Yaskawa INFORM job: R1_W27-A2(70,-90)ZJEBANY.JBI

/JOB
//NAME R1_W27-A2(70,-90)ZJEBANY
///FOLDERNAME KRIS-SCIANA
//POS
///NPOS 112,112,0,3,0,0
///TOOL 0
///POSTYPE PULSE
///PULSE
C00000=15585,66998,-23352,-10992,101775,82043
C00001=-39674,-71250,-76076,2670,72414,70019
C00002=-101235,-135701,-102906,17581,29400,53654
C00003=-127456,-117366,-93315,32899,50159,54489
C00004=-154723,-66087,-38493,57483,73854,47255
C00005=-151694,-18406,22661,89573,79243,43877
C00006=-147945,-16802,25938,90973,76715,43351
C00007=-146442,-16053,27339,91568,75716,43130
C00008=-145555,-16531,26989,91866,75130,43118
C00009=-146442,-16053,27339,91568,75716,43130
C00010=-129825,-25208,-16895,45276,72510,50220
C00011=-129825,-26937,-23175,44700,74652,51212
C00012=-126968,34908,31795,39712,91911,59385
C00013=-127089,30774,28423,39703,91929,59340
C00014=-127131,29285,26942,39705,92062,59372
C00015=-126987,33781,29619,39748,92512,59603
C00016=-124782,21409,16268,39949,92944,60731
C00017=-124782,21545,16842,39933,92724,60648
C00018=-124794,21102,17061,39913,92450,60538
C00019=-124782,20683,12912,40055,94258,61228
C00020=-126312,48107,49635,39662,88339,58341
C00021=-126284,49606,51426,39664,88067,58253
C00022=-126313,48129,49805,39664,88266,58315
C00023=-132184,54704,68476,52529,88046,54125
C00024=-131484,54267,67976,52659,87709,54297
C00025=-125376,45201,47158,39737,87937,58598
C00026=-125376,43761,43100,39745,89306,59110
C00027=-123484,43447,42766,39862,88476,59619
C00028=-123496,42639,42608,39862,88236,59522
C00029=-123484,43447,42766,39862,88476,59619
C00030=-128193,-56545,-35379,53218,50640,50358
C00031=-130143,-61631,-36192,55096,50491,48856
C00032=-129949,-27153,-29048,38459,86720,4249
C00033=-121863,7196,-1024,23892,106167,-36201
C00034=-119790,7803,2418,24012,103908,-35875
C00035=-119251,9137,4734,24063,102944,-35747
C00036=-119851,8106,3844,23917,103264,-36033
C00037=-118959,8581,3089,24147,103654,-35610
C00038=-119216,9443,7897,23894,101312,-36052
C00039=-119770,8589,6030,23811,102232,-36216
C00040=-121844,7811,2421,23662,104503,-36541
C00041=-94529,-5213,-25149,-6002,99872,9031
C00042=-100194,-9058,-21367,-2473,91495,-15305
C00043=-91351,-8865,-21769,-5973,96170,10290
C00044=-91796,-6310,-20482,-5976,96656,10116
C00045=-96950,-9343,-21983,-4178,92826,-6406
C00046=-96879,-9292,-21943,-4182,92831,-6382
C00047=-95506,-8282,-21147,-4258,92931,-5923
C00048=-95506,-8333,-22847,-4265,93948,-5958
C00049=-93861,17350,-1887,-1756,103785,47914
C00050=-93642,17646,1086,-1725,102113,48015
C00051=-99387,63034,56242,88,91722,55973
C00052=-99595,65462,59338,72,91065,55902
C00053=-107274,85511,83456,10826,96806,70956
C00054=-106567,101770,109831,10934,91162,70697
C00055=-107923,97580,104079,9794,92669,70451
C00056=-108057,102398,108554,9757,92409,70386
C00057=-105555,82062,76147,4864,95020,72280
C00058=-105152,38520,-21397,2190,99545,72640
C00059=-7518,84886,-13149,67305,106234,67756
C00060=22775,131727,30764,-8837,96794,84364
C00061=11815,113566,24775,-13722,103628,75456
C00062=-62332,57779,42971,-10705,100391,40003
C00063=-63598,57661,46336,-10776,98127,39757
C00064=-59832,79873,78506,-18224,98168,41291
C00065=-60139,78050,76254,-18318,98529,41127
C00066=-64108,57720,47808,-10808,97198,39660
C00067=-61440,56043,48331,-17001,92681,37273
C00068=-61968,56499,48847,-17036,92491,37113
C00069=-61419,54058,46112,-17010,93016,37234
C00070=-68170,68334,55591,-4501,100736,41870
C00071=-70059,62116,48331,-4828,101895,41166
C00072=-69967,61865,48814,-4804,101477,41214
C00073=-70059,62116,48331,-4828,101895,41166
C00074=-68170,68334,55591,-4501,100736,41870
C00075=-66509,67398,53143,-4253,101849,42410
C00076=-80402,67204,62355,-14177,107743,50421
C00077=-80401,69312,67811,-13985,105535,50686
C00078=-80884,69661,69168,-14085,104811,50596
C00079=-80514,70324,68988,-14005,105317,50671
C00080=-79798,72099,72356,-13691,104310,51048
C00081=-81157,88532,95788,-17232,96100,47498
C00082=-80402,71338,72587,-13845,103689,50903
C00083=-80402,69349,67894,-13982,105503,50690
C00084=-64491,51473,31572,1240,90356,18022
C00085=-65162,54788,38997,1284,87502,17767
C00086=-65274,58172,43940,1291,86202,17717
C00087=-65583,56675,41439,1312,86976,17619
C00088=-64984,54297,39530,1273,86918,17821
C00089=-65111,58482,44265,1282,86158,17770
C00090=-64897,62335,49011,1268,85210,17834
C00091=-65160,54781,38996,1284,87498,17768
C00092=-64488,51465,31572,1240,90352,18023
C00093=-66978,64834,55479,27147,84077,-20274
C00094=-66978,66406,60274,27238,82160,-20721
C00095=-66806,67592,62294,27265,81538,-20800
C00096=-67518,65114,59942,27279,81926,-20981
C00097=-67126,67247,61249,27252,82058,-20801
C00098=-67182,73036,74425,27621,77495,-21906
C00099=-66978,71231,72456,27590,77681,-21782
C00100=-66977,69736,68964,27473,78911,-21487
C00101=-107213,71290,72523,349,112834,-78845
C00102=-107215,71286,72519,348,112835,-78845
C00103=-106198,74490,76377,813,112100,-78474
C00104=-107250,71387,71410,334,113570,-78856
C00105=-107326,75265,77802,294,111629,-78889
C00106=-107814,73110,74567,72,112512,-79066
C00107=-107214,71283,72515,348,112836,-78845
C00108=-107213,71286,72519,349,112835,-78845
C00109=-107166,72243,73362,386,91253,-78825
C00110=-107166,72243,73362,386,91253,-78825
C00111=-63792,102119,73362,386,91253,666
BC00000=173361,170327,1069948
BC00001=285044,126360,1057855
BC00002=365463,938,1004473
BC00003=471,4089,1024902
BC00004=269,7512,1047096
BC00005=15,11820,1075020
BC00006=15,11820,1075020
BC00007=15,11820,1075020
BC00008=15,11820,1075020
BC00009=15,11820,1075020
BC00010=15,11820,1075020
BC00011=15,11820,1075020
BC00012=15,11820,1075020
BC00013=15,11820,1075020
BC00014=15,11821,1075019
BC00015=15,11820,1075020
BC00016=15,11820,1075020
BC00017=15,11820,1075020
BC00018=15,11820,1075020
BC00019=15,11820,1075020
BC00020=15,11820,1075020
BC00021=15,11820,1075020
BC00022=15,11820,1075020
BC00023=15,11820,1075020
BC00024=15,11820,1075020
BC00025=15,11820,1075020
BC00026=15,11820,1075020
BC00027=15,11820,1075020
BC00028=15,11820,1075020
BC00029=15,11820,1075020
BC00030=15,11820,1075020
BC00031=15,11820,1075020
BC00032=15,31624,1075102
BC00033=15,49099,1075175
BC00034=15,47849,1075175
BC00035=15,47349,1075175
BC00036=15,47349,1075175
BC00037=15,47349,1075175
BC00038=15,62077,1075175
BC00039=15,62577,1075175
BC00040=15,63827,1075175
BC00041=15,12213,1075175
BC00042=16,12213,1075171
BC00043=15,16755,1075175
BC00044=15,16755,1075175
BC00045=16,12213,1075171
BC00046=16,12213,1075171
BC00047=16,12213,1075171
BC00048=16,12213,1075171
BC00049=16,12213,1075171
BC00050=16,12213,1075171
BC00051=16,12213,1075171
BC00052=16,12213,1075171
BC00053=17,22433,1075169
BC00054=17,22433,1075167
BC00055=17,22433,1075169
BC00056=17,22433,1075169
BC00057=16,12213,1075171
BC00058=16,12213,1075171
BC00059=25030,15919,1060143
BC00060=103306,16446,1075157
BC00061=154602,14134,1075161
BC00062=246913,5043,1075175
BC00063=246913,5043,1075175
BC00064=246913,5043,1075175
BC00065=246913,5043,1075175
BC00066=246913,5043,1075175
BC00067=246913,5043,1075175
BC00068=246913,5043,1075175
BC00069=246913,5043,1075175
BC00070=246913,5043,1075175
BC00071=246913,5043,1075175
BC00072=246913,5043,1075175
BC00073=246913,5043,1075175
BC00074=246913,5043,1075175
BC00075=246913,5043,1075175
BC00076=310215,25331,1075175
BC00077=304559,24148,1075175
BC00078=304559,24148,1075175
BC00079=302296,23674,1075175
BC00080=302296,23674,1075175
BC00081=304559,24148,1075175
BC00082=304613,38875,1070974
BC00083=310269,40059,1075175
BC00084=197323,15,1075175
BC00085=197986,15,1075175
BC00086=197986,15,1075175
BC00087=198252,15,1075175
BC00088=198252,15,1075175
BC00089=200364,15,1075175
BC00090=200364,15,1075175
BC00091=200098,15,1075175
BC00092=199434,15,1075175
BC00093=148787,33401,1075175
BC00094=154351,32151,1075175
BC00095=156150,31747,1075172
BC00096=156576,31651,1075175
BC00097=156576,31651,1075175
BC00098=156716,69750,1059420
BC00099=154490,70250,1066913
BC00100=148927,71500,1075175
BC00101=344706,64580,1052547
BC00102=343940,58320,1037184
BC00103=343634,55816,1031039
BC00104=343634,55816,1031039
BC00105=343634,55816,1031039
BC00106=343634,55816,1031039
BC00107=340873,58338,1037257
BC00108=341638,64598,1052619
BC00109=341637,64597,1052617
BC00110=398183,64597,1052617
BC00111=370823,64597,1052617
///POSTYPE BASE
///RECTAN
///RCONF 0,0,0,0,1,0,0,0,0,0,0,0,0,0,0,0,0,0,0,0,0,0,0,0
P00006=2.006,1.622,-0.565,0.0000,0.0000,0.0000
///RCONF 0,0,0,0,0,0,0,0,0,0,0,0,0,0,0,0,0,0,0,0,0,0,0,0
P00023=-2.957,-4.083,2.762,0.0000,0.0000,0.0000
P00024=-1.466,-0.226,-0.419,0.0000,0.0000,0.0000
//INST
///DATE 2023/12/05 17:02
///ATTR SC,RW
///GROUP1 RB1,BS1
NOP
'r1_W27-A2(70,-90)
'Path S987
SFTOF
MOVJ C00000 BC00000 VJ=100.00
MOVJ C00001 BC00001 VJ=100.00
MOVJ C00002 BC00002 VJ=100.00
MOVJ C00003 BC00003 VJ=100.00
MOVJ C00004 BC00004 VJ=70.00
MOVJ C00005 BC00005 VJ=100.00
MOVJ C00006 BC00006 VJ=100.00
MOVL C00007 BC00007 V=60.0
REFP 3 C00008 BC00008
CALL JOB:SEARCH-R1
SET P023 P006
SFTON P023
MOVL C00009 BC00009 V=60.0
MOVL C00010 BC00010 V=60.0
MOVL C00011 BC00011 V=60.0
MOVL C00012 BC00012 V=60.0
MOVL C00013 BC00013 V=60.0
REFP 3 C00014 BC00014
CALL JOB:SEARCH-R1
SET P023 P006
SFTON P023
MOVL C00015 BC00015 V=60.0
MOVL C00016 BC00016 V=60.0
MOVL C00017 BC00017 V=100.0
REFP 3 C00018 BC00018
CALL JOB:SEARCH-R1
SET P023 P006
SFTON P023
MOVL C00019 BC00019 V=60.0
'DRUGI NOWY POMIAR
SFTOF
MOVL C00020 BC00020 V=60.0
REFP 3 C00021 BC00021
CALL JOB:SEARCH-R1
SET P024 P006
SFTON P024
MOVL C00022 BC00022 V=60.0
MOVL C00023 BC00023 V=60.0
REFP 3 C00024 BC00024
CALL JOB:SEARCH-R1
SET P024 P006
SFTON P024
MOVL C00025 BC00025 V=60.0
MOVL C00026 BC00026 V=60.0
MOVL C00027 BC00027 V=60.0
REFP 3 C00028 BC00028
CALL JOB:SEARCH-R1
SET P024 P006
SFTON P024
MOVL C00029 BC00029 V=60.0
MOVL C00030 BC00030 V=100.0
MOVL C00031 BC00031 V=1000.0
'Path VIA1118
SFTOF
MOVJ C00032 BC00032 VJ=100.00
'Path W988
SFTOF
SFTON P023
MOVJ C00033 BC00033 VJ=100.00
MOVJ C00034 BC00034 VJ=100.00
MOVL C00035 BC00035 V=100.0 PL=0
REFP 1 C00036 BC00036
REFP 2 C00037 BC00037
MACRO1 MJ#(0) ARGF7
ARCON
SFTON P024
MOVL C00038 BC00038 V=11.5
ARCOF
MOVL C00039 BC00039 V=100.0
MOVL C00040 BC00040 V=166.7
SFTOF
'Path W989
SFTOF
SFTON P023
MOVJ C00041 BC00041 VJ=100.00
MOVL C00042 BC00042 V=100.0 PL=0
REFP 1 C00043 BC00043
REFP 2 C00044 BC00044
MACRO1 MJ#(0) ARGF7
ARCON
MOVL C00045 BC00045 V=11.7
MOVL C00046 BC00046 V=11.7
MOVL C00047 BC00047 V=11.7
ARCOF
MOVJ C00048 BC00048 VJ=100.00
MOVJ C00049 BC00049 VJ=100.00
MOVJ C00050 BC00050 VJ=100.00
ARCON
SFTON P024
MOVL C00051 BC00051 V=11.7
MOVL C00052 BC00052 V=11.7
ARCOF
MOVJ C00053 BC00053 VJ=100.00
MOVJ C00054 BC00054 VJ=100.00
ARCON
MOVL C00055 BC00055 V=11.7
ARCOF
MOVL C00056 BC00056 V=100.0
MOVL C00057 BC00057 V=166.7
MOVJ C00058 BC00058 VJ=100.00
SFTOF
'2 STRONA
MOVJ C00059 BC00059 VJ=100.00
'Path VIA1124
SFTOF
MOVJ C00060 BC00060 VJ=100.00
CALL JOB:ONLYCUT-R1_LONG
'Path S992
SFTOF
MOVJ C00061 BC00061 VJ=100.00
MOVJ C00062 BC00062 VJ=100.00
MOVJ C00063 BC00063 VJ=100.00
MOVL C00064 BC00064 V=60.0
REFP 3 C00065 BC00065
CALL JOB:SEARCH-R1
SET P024 P006
SFTON P024
MOVL C00066 BC00066 V=60.0
MOVL C00067 BC00067 V=60.0
REFP 3 C00068 BC00068
CALL JOB:SEARCH-R1
SET P024 P006
SFTON P024
MOVL C00069 BC00069 V=60.0
MOVL C00070 BC00070 V=100.0
MOVL C00071 BC00071 V=60.0
REFP 3 C00072 BC00072
CALL JOB:SEARCH-R1
SET P024 P006
SFTON P024
MOVL C00073 BC00073 V=60.0
MOVL C00074 BC00074 V=100.0
MOVL C00075 BC00075 V=166.7
'Path W993
SFTOF
SFTON P024
MOVJ C00076 BC00076 VJ=100.00
MOVJ C00077 BC00077 VJ=100.00
MOVL C00078 BC00078 V=100.0 PL=0
REFP 1 C00079 BC00079
REFP 2 C00080 BC00080
MACRO1 MJ#(0) ARGF7
ARCON
MOVL C00081 BC00081 V=11.5
ARCOF
MOVL C00082 BC00082 V=100.0
MOVL C00083 BC00083 V=166.7
SFTOF
'Path W994
SFTOF
SFTON P024
MOVJ C00084 BC00084 VJ=100.00
MOVJ C00085 BC00085 VJ=100.00
MOVL C00086 BC00086 V=100.0 PL=0
REFP 1 C00087 BC00087
REFP 2 C00088 BC00088
MACRO1 MJ#(0) ARGF7
ARCON
MOVL C00089 BC00089 V=11.5
MOVL C00090 BC00090 V=11.7
ARCOF
MOVL C00091 BC00091 V=100.0
MOVL C00092 BC00092 V=166.7
SFTOF
'Path W995
SFTOF
SFTON P024
MOVJ C00093 BC00093 VJ=100.00
MOVJ C00094 BC00094 VJ=100.00
MOVL C00095 BC00095 V=100.0 PL=0
REFP 1 C00096 BC00096
REFP 2 C00097 BC00097
MACRO1 MJ#(0) ARGF7
ARCON
MOVL C00098 BC00098 V=11.5
ARCOF
MOVL C00099 BC00099 V=400.0
MOVL C00100 BC00100 V=1000.0
SFTOF
'Path W996
SFTOF
SFTON P024
MOVJ C00101 BC00101 VJ=100.00
MOVJ C00102 BC00102 VJ=100.00
MOVL C00103 BC00103 V=100.0 PL=0
REFP 1 C00104 BC00104
REFP 2 C00105 BC00105
MACRO1 MJ#(0) ARGF7
ARCON
MOVL C00106 BC00106 V=11.5
ARCOF
MOVL C00107 BC00107 V=100.0
MOVL C00108 BC00108 V=166.7
SFTOF
MOVJ C00109 BC00109 VJ=100.00
MOVJ C00110 BC00110 VJ=80.00
MOVJ C00111 BC00111 VJ=80.00
'obrot
END
